Omron CX-Programmer project NewProject (CX-Programmer 9.03)

# PLC NewPLC1: CP1L L

## Global symbols (name address type ; comment)
0.00 BOOL  ; Switch a
0.01 BOOL  ; Switch b
1.00 BOOL  ; lampu

## Program NewProgram1 (cyclic task 0)

### Section Section1

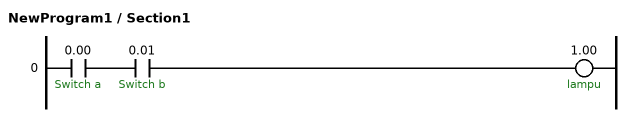
; rung 0
LD 0.00  ; Switch a
AND 0.01  ; Switch b
OUT 1.00  ; lampu

### Section END
; rung 0
END(001)